{attribute 'no_check'}
FUNCTION_BLOCK OUTPUT
VAR_INPUT
	EN														:	BOOL := TRUE;
	IN														:	BOOL := FALSE;
END_VAR         								
VAR_OUTPUT      								
	status													:	BYTE := 0;
	Q												AT  %Q* :	BOOL;
END_VAR         							
VAR             				
END_VAR

IF IN THEN
	ON();
ELSE
	OFF();
END_IF

status.0 													:= NOT Q;
status.1 													:= Q;
status.5 													:= NOT EN;

METHOD PUBLIC OFF
VAR_INPUT
END_VAR
Q															:= IN := FALSE;
END_METHOD

METHOD PUBLIC ON
VAR_INPUT
END_VAR
IN 															:= TRUE;
Q 															:= EN AND IN;
END_METHOD

END_FUNCTION_BLOCK

(* stored: Version 1.1.0.1, ProductVersion 3.1.4024.12
   POU OUTPUT: Id {bfc4f4e5-dbe0-41dd-9de3-68ac105cf38e}, SpecialFunc None
   Method OFF: Id {7a803ce3-62fc-4d11-b256-e7afcdaa7d24}
   Method ON: Id {d845a3e4-f40a-4cb9-89a0-c12196b98144} *)
